FUNCTION_BLOCK FB_analo_and_digital
VAR_INPUT
	iRAWValue : LREAL;			//raw Value read from sensor (registre)
	iResolution : INT; 		//resolution in bits
	iValMin: INT;			//min physical value possible
	iValMax: INT;			//max physical value possible
	iTransToPhysical : BOOL;	//RAW --> Physical when TRUE
	iPhysical2Value: LREAL; 	//valeur physique (ex tr/min)
	iValInputMax: INT;		//max input value at the Box
	iValInputMin: INT;		//min input value at the Box
	iPhysicalValue : LREAL;	//valeur physique sur l'entree de l'input
END_VAR
VAR_OUTPUT
	oValInputMin: INT;		//min input value at the Box
	oPhysicalValue : LREAL;	//valeur physique sur l'entree de l'input
	oInputValue : LREAL;	//valeur physique sur l'entree de l'input
	oPhysical2Value: LREAL; 	//valeur physique (ex tr/min)
	oRAWValue : LREAL;			//raw Value read from sensor (registre)
END_VAR
VAR	
	temp : LREAL;
	temp2 : LREAL;	
END_VAR

temp2:=expt(2,iResolution);



IF(iTransToPhysical) THEN
	//RAW Input to physical value
	temp:=(iValInputMax-iValInputMin) / temp2;
	oInputValue:=iValInputMin + (temp * (iRAWValue + temp2/2));
	
	
	temp:=(iValMax-iValMin) / temp2;
	oPhysicalValue:=iValMin + (temp * (iRAWValue+temp2/2));
ELSE
	//Physical value to raw-Value
	temp:=(iValMax-iValMin) / temp2;
	oRAWValue:= iValMin+ (iPhysicalValue / temp);
			
END_IF

END_FUNCTION_BLOCK

(* stored: Version 1.1.0.1, ProductVersion 3.1.4020.6
   POU FB_analo_and_digital: Id {2e0b3f33-2d6e-4edd-9bfd-609786c9e06f}, SpecialFunc None *)
